{attribute 'qualified_only'}
{attribute 'strict'}
TYPE E_Z2_Step :
(
	(* special steps *)
	NoStep := -32767,		// nessuno step
	Unknown := -32000,		// step sconosciuto
	
	(* Error steps *)
	NeOrError := -990,		// non abilitata o in errore
	Recovering := -980,		// azzeramento errori
		
	(* Stop *)
	Stop := 0,				// S0, stop
	
	(* Cycle *)
	Ready := 100,			// S1, pronto a ricevere pezzo
	WaitZ3Ready := 120,		// S2, aspetta che Z3 sia libera
	MoveForward := 140,		// S3, trasferimento pezzo verso Z2 
	MoveBackward := 160,	// S4, ritorno slitta

	Done := 800,			// Ciclo concluso
	
	(* Stopping *)
	Stopping := 900	
);
END_TYPE
//  NoStep = '-32767'
//  Unknown = '-32000'
//  NeOrError = '-990'
//  Recovering = '-980'

(* stored: Version 1.1.0.1
   EnumerationTextList E_Z2_Step: Id {d49f30c0-3193-0e23-2037-f633790ab29c} *)
